// TIA Portal V19 export
DATA_BLOCK "InfeedPAC3200_Adv"   // DB36
TITLE = Instance DB of advanced energy data collection
// Instance DB of advanced energy data collection
// stored: InstanceOfName EnS_EnergyDataAdv, InstanceOfType FB
"EnS_EnergyDataAdv"
   // VAR_INPUT
   //    advData { ExternalWritable := 'False'} : "EnS_typeEnergyAdv";
   // END_VAR
   // VAR_OUTPUT
   //    error { ExternalAccessible := 'False'; ExternalVisible := 'False'; ExternalWritable := 'False'} : Bool;
   //    status { ExternalAccessible := 'False'; ExternalVisible := 'False'; ExternalWritable := 'False'} : Word;
   // END_VAR
   // VAR_IN_OUT
   //    orgData : "EnS_typeOrgData";
   //    energyMeta : "EnS_typeEnergyMeta";
   // END_VAR
BEGIN
END_DATA_BLOCK
